// SIMATIC S7-200 project (STEP 7-Micro/WIN), CPU 221 REL 01.10

SYMBOL_TABLE USER1
CD2              M0.1
CD1              M0.0
ONN1             I0.0
OFF              I0.2
DEN              Q0.0
ONN2             I0.1
END_SYMBOL_TABLE

ORGANIZATION_BLOCK MAIN:OB1
TITLE=PROGRAM COMMENTS
BEGIN
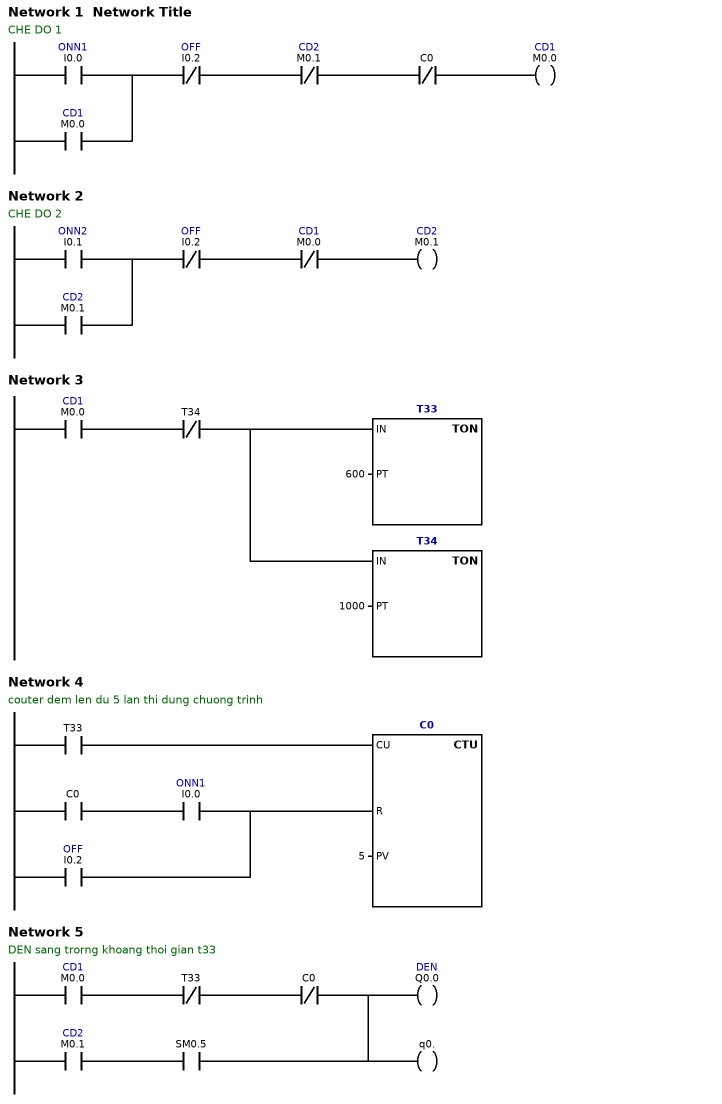
Network 1 // Network Title
// CHE DO 1
LD     ONN1:I0.0
O      CD1:M0.0
AN     OFF:I0.2
AN     CD2:M0.1
AN     C0
=      CD1:M0.0
Network 2
// CHE DO 2
LD     ONN2:I0.1
O      CD2:M0.1
AN     OFF:I0.2
AN     CD1:M0.0
=      CD2:M0.1
Network 3
LD     CD1:M0.0
AN     T34
TON    T33, 600
TON    T34, 1000
Network 4
// couter dem len du 5 lan thi dung chuong trinh
LD     T33
LD     C0
A      ONN1:I0.0
O      OFF:I0.2
CTU    C0, 5
Network 5
// DEN sang trorng khoang thoi gian t33
// (network saved uncompiled; LAD cells follow)
// row 0: c0 -| |- CD1:M0.0  c1 -|/|- T33  c2 -|/|- C0 v  c3 -( ) DEN:Q0.0
// row 1: c0 -| |- CD2:M0.1  c1 -| |- SM0.5  c2 -- ^  c3 -( ) q0.
END_ORGANIZATION_BLOCK
